INTERFACE I_MessageData

PROPERTY DirRoot : POINTER to string(255)
SET
END_SET
END_PROPERTY

PROPERTY ErrorIndex : reference to uint
SET
END_SET
END_PROPERTY

PROPERTY FileRoot : pointer to string(255)
SET
END_SET
END_PROPERTY

PROPERTY LocalTime : pointer to DT
SET
END_SET
END_PROPERTY

PROPERTY MessageIndex : reference to uint
SET
END_SET
END_PROPERTY

PROPERTY MsgList : pointer to ARRAY[1..GVL_MSG.MAX_MESSAGE] OF st_message
SET
END_SET
END_PROPERTY

END_INTERFACE

(* stored: Version 1.1.0.1
   Itf I_MessageData: Id {aed2e1ec-9d55-41ea-a69f-e049e51a742c}
   Property DirRoot: Id {4ca21754-ac5d-43f1-bbad-65cd7f5f4ff2}
   Set Set: Id {cfaddee8-59a2-4795-a3ef-71fa67f89ca5}
   Property ErrorIndex: Id {24a0c1c6-ded5-4a3f-ae24-fe85b7e8f46b}
   Set Set: Id {b06166be-c73d-4507-a5b1-a7f57394221a}
   Property FileRoot: Id {4ad4f349-d2c9-40ca-9f08-d0c5127cbf4f}
   Set Set: Id {6a732649-2105-412b-a170-7d3cbc5b32c4}
   Property LocalTime: Id {30af9ab5-de00-41c6-8568-30529e779254}
   Set Set: Id {22e7aa6d-1323-4e38-af05-3ca2629d3abc}
   Property MessageIndex: Id {92a6a32b-eb2f-4c36-a349-cef6e5ebd756}
   Set Set: Id {224b5733-9739-4951-91ed-14ce77c26366}
   Property MsgList: Id {8af2c207-ee0c-4636-bcf3-930cee315713}
   Set Set: Id {71c4b180-c9c1-4c0c-8a55-25757d4c3dd8} *)
